Universal Robots PolyScope program: punto3_pickplace.urp

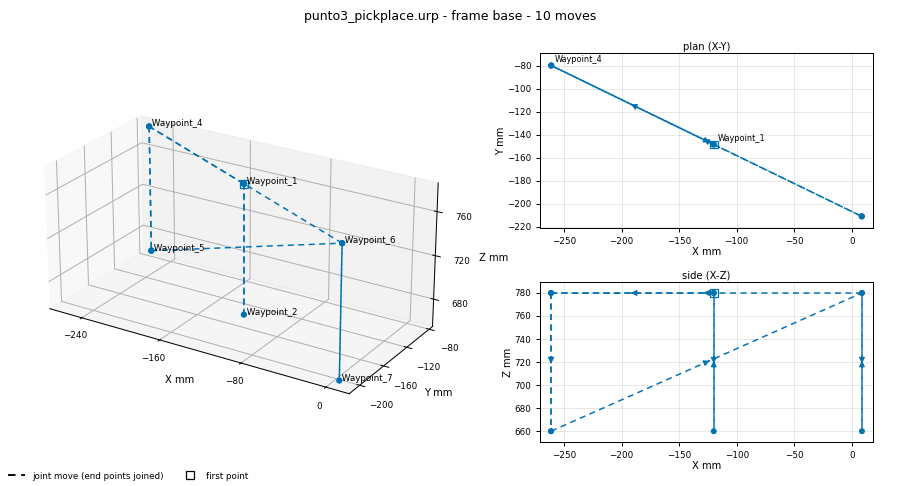
[picture p0: tool path of punto3_pickplace.urp in frame base, 10 of 10 moves have a stored position in this frame; points joined in program order, loops and branches not executed]
Program punto3_pickplace (installation=default directory=/ursim/programs createdIn=3.15.8.106339 lastSavedIn=3.15.8.106339 robotSerialNumber=2018359999)
Calibrated DH parameters: a=[0, -0.425, -0.39225, 0, 0, 0]; d=[0.089159, 0, 0, 0.10915, 0.09465, 0.0823]; alpha=[1.570796, 0, 0, 1.570796, -1.570796, 0]; deltaTheta=[0, 0, 0, 0, 0, 0]
Robot Program (runOnlyOnce=false)
  MoveJ speed 60 deg/s, acceleration 80 deg/s^2 (useActiveTCP=true)
    Set DigitalOutput pin=digital_out[0]; digitalValue=0
    Waypoint Waypoint_1: TCP in base x=-119.94 y=-148.524 z=780 mm, rx=-0.0392 ry=2.2037 rz=-2.2037 rad; joints [-23.094, -41.258, -85.091, -53.651, 25.118, -0.012] deg
    Waypoint Waypoint_2: TCP in base x=-119.94 y=-148.524 z=660 mm, rx=-0.0392 ry=2.2037 rz=-2.2037 rad; joints [-100.212, -49.741, -107.482, -22.778, 102.236, -0.012] deg
    Set DigitalOutput pin=digital_out[0]; digitalValue=1
    Popup Message (haltProgram=false message=se cerró el gripper  inputType=Text)
    Waypoint Waypoint_3: TCP in base x=-119.94 y=-148.524 z=780 mm, rx=-0.0392 ry=2.2037 rz=-2.2037 rad; joints [-23.094, -41.258, -85.091, -53.651, 25.118, -0.012] deg
    Popup Message (haltProgram=false message=punto intermedio inputType=Text)
    Wait Sleep waitTime=1
    Waypoint Waypoint_4: TCP in base x=-261.164 y=-79.932 z=780 mm, rx=-0.0392 ry=2.2037 rz=-2.2037 rad; joints [-24.916, -31.672, -76.332, -71.996, 26.94, -0.012] deg
    Popup Message (haltProgram=false message=punto intermedio llegada inputType=Text)
    Waypoint Waypoint_5: TCP in base x=-261.164 y=-79.932 z=660 mm, rx=-0.0392 ry=2.2037 rz=-2.2037 rad; joints [-156.089, -70.157, -98.608, -11.235, 158.113, -0.012] deg
    Set DigitalOutput pin=digital_out[0]; digitalValue=0
    Popup Message (haltProgram=false message=se abrió el gripper inputType=Text)
    Wait Sleep waitTime=1
    Waypoint Waypoint_6: TCP in base x=8.691 y=-210.999 z=780 mm, rx=-0.0392 ry=2.2037 rz=-2.2037 rad; joints [-29.55, -55.888, -85.587, -38.525, 31.574, -0.012] deg
    Set DigitalOutput pin=digital_out[0]; digitalValue=0
    Waypoint Waypoint_7: TCP in base x=8.691 y=-210.999 z=660 mm, rx=-0.0392 ry=2.2037 rz=-2.2037 rad; joints [-29.55, -47.346, -108, -24.654, 31.574, -0.012] deg
    Set DigitalOutput pin=digital_out[0]; digitalValue=1
    Popup Message (haltProgram=false message=se cerró el gripper inputType=Text)
    Waypoint Waypoint_8: TCP in base x=8.691 y=-210.999 z=780 mm, rx=-0.0392 ry=2.2037 rz=-2.2037 rad; joints [-29.55, -55.888, -85.587, -38.525, 31.574, -0.012] deg
    Popup Message (haltProgram=false message=punto intermedio inputType=Text)
    Wait Sleep waitTime=1
    Waypoint Waypoint_9: TCP in base x=-261.164 y=-79.932 z=780 mm, rx=-0.0392 ry=2.2037 rz=-2.2037 rad; joints [-24.916, -31.672, -76.332, -71.996, 26.94, -0.012] deg
    Waypoint Waypoint_10: TCP in base x=-261.164 y=-79.932 z=660 mm, rx=-0.0392 ry=2.2037 rz=-2.2037 rad; joints [-156.089, -70.157, -98.608, -11.235, 158.113, -0.012] deg
    Set DigitalOutput pin=digital_out[0]; digitalValue=0
    Popup Message (haltProgram=false message=se abrió el gripper inputType=Text)
    Wait Sleep waitTime=1
    Wait DigitalInput pin=digital_in[0]; digitalValue=1
